# EPICS autosave request: iocBoot/gmca_23i_ioc1/dbSave/BD_DhB_.req
%
% BURT Request File
%
% $(P)BD:DhB: Horizontal Beam Delivery for BM line (type: XPs)
%

file assy.req ASSY=$(P)BD:DhB
file mtr1.req MTR1=$(P)BD:mhd
file drv1.req DRV1=$(P)BD:HD
